// Mitsubishi GX Works2 project: PLC 적산 타이머, 카운터 예제 1   PLC: Q03UDV

PROGRAM MAIN
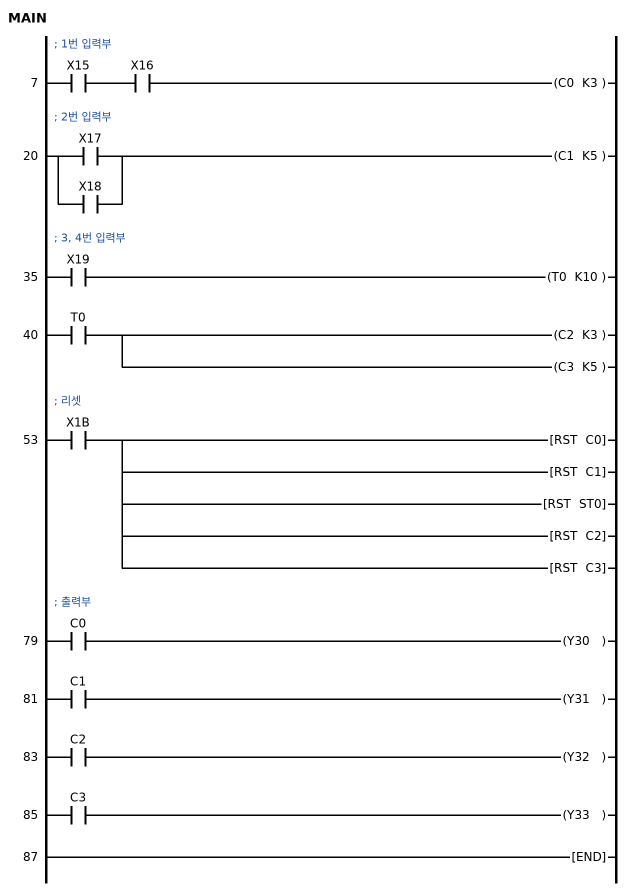
; 1번 입력부
7     LD      X15
      AND     X16
      OUT     C0 K3
; 2번 입력부
20    LD      X17
      OR      X18
      OUT     C1 K5
; 3, 4번 입력부
35    LD      X19
      OUT     T0 K10
40    LD      T0
      OUT     C2 K3
      OUT     C3 K5
; 리셋
53    LD      X1B
      RST     C0
      RST     C1
      RST     ST0
      RST     C2
      RST     C3
; 출력부
79    LD      C0
      OUT     Y30
81    LD      C1
      OUT     Y31
83    LD      C2
      OUT     Y32
85    LD      C3
      OUT     Y33
87    END
END_PROGRAM
